// TIA Portal V19 export
DATA_BLOCK "A0301_PTrk_To_BTrk_Create"   // DB183
// stored: InstanceOfName A0301_PTrk_To_BTrk_Create_FB, InstanceOfType FB
"A0301_PTrk_To_BTrk_Create_FB"
   // VAR_INPUT
   //    AreaInterface : "AreaInterface";
   //    Execute : Bool;
   //    PTrk_P2 { ExternalAccessible := 'False'; ExternalVisible := 'False'; ExternalWritable := 'False'} : "PTrk_Item";
   //    PTrk_P3 { ExternalAccessible := 'False'; ExternalVisible := 'False'; ExternalWritable := 'False'} : "PTrk_Item";
   // END_VAR
   // VAR_OUTPUT
   //    BTrk { ExternalAccessible := 'False'; ExternalVisible := 'False'; ExternalWritable := 'False'} : "BTrk_item";
   // END_VAR
   // VAR_IN_OUT
   //    Status : USInt;
   // END_VAR
   // VAR
   //    R_TRIG_Execute { S7_SetPoint := 'True'} : R_TRIG;
   //    Inc_Last_ID_B { ExternalAccessible := 'False'; ExternalVisible := 'False'; ExternalWritable := 'False'} : Bool;
   //    Alarm { ExternalAccessible := 'False'; ExternalVisible := 'False'; ExternalWritable := 'False'} : USInt;
   // END_VAR
BEGIN
END_DATA_BLOCK
